// TIA Portal V19 export
DATA_BLOCK "LB211"   // DB145
// stored: InstanceOfName ButtonsSafe_LB211, InstanceOfType FB
"ButtonsSafe_LB211"
   // VAR_INPUT
   //    Reset_OthersPBs_Activation_IN : Bool;
   // END_VAR
   // VAR_OUTPUT
   //    Reset_OthersPBs_Activation_OUT : Bool;
   // END_VAR
   // VAR
   //    SelectionIs_Bwd : Bool;
   //    SelectionIs_Fwd : Bool;
   //    Pb_PEAux : Bool;
   //    PB : Struct
   //       ResetAlarms : Bool;
   //       Rollformer_Bwd : Bool;
   //       Rollformer_Fwd : Bool;
   //    END_STRUCT;
   // END_VAR
BEGIN
END_DATA_BLOCK
